INTERFACE ICommunicationRoboterOmron EXTENDS __SYSTEM.IQueryInterface

METHOD ContactPrepared
VAR_INPUT
    enable : BOOL;
END_VAR
END_METHOD

PROPERTY EState : E_SocketConnectionState
GET
END_GET
END_PROPERTY

METHOD HighPowerOn
VAR_INPUT
    enable : BOOL;
END_VAR
END_METHOD

PROPERTY MsgFmtStr : T_MaxString
GET
END_GET
END_PROPERTY

METHOD RequestHome
VAR_INPUT
    enable : BOOL;
END_VAR
END_METHOD

METHOD Reset
VAR_INPUT
    enable : BOOL;
END_VAR
END_METHOD

METHOD Run
END_METHOD

METHOD StartAutomatic
VAR_INPUT
    enable : BOOL;
END_VAR
END_METHOD

METHOD StopAutomatic
VAR_INPUT
    enable : BOOL;
END_VAR
END_METHOD

END_INTERFACE

(* stored: Version 1.1.0.1, ProductVersion 3.1.4024.12
   Itf ICommunicationRoboterOmron: Id {996aedc9-c4c3-0ece-1bac-eb0c3ba8695f}
   Folder Commands: Id {d1ee2977-2e1d-0c9a-1f8d-700840bf107a}
   Method ContactPrepared: Id {e2a4f042-87e0-09a8-2516-ac045da79c2a}
   Property EState: Id {a554bf8d-3668-0bf6-2ebb-f98b68de1bb5}
   Get Get: Id {c3d60dbf-a4c4-070d-2af6-c7e47b26ba7a}
   Method HighPowerOn: Id {65a7d103-5df9-01df-1cd2-b3e4db9fc1b1}
   Property MsgFmtStr: Id {17a091ed-baf9-04c0-129a-d545380b55db}
   Get Get: Id {0fce75c3-e9f4-09bd-0737-52dd852a93b7}
   Method RequestHome: Id {6d38cf01-0273-02f2-3f63-50cd1db295c6}
   Method Reset: Id {4ef9796b-6ba3-0cf1-0d22-83fcd722b75d}
   Method Run: Id {558e231b-2dc8-0ccc-29ab-5a99bfe9691b}
   Method StartAutomatic: Id {55967697-6e1c-0795-170c-95595c3068ad}
   Method StopAutomatic: Id {afa72e8f-f0d8-0233-0dce-2733ed2fe2b1} *)
